// TIA Portal V21 export
ORGANIZATION_BLOCK "Cyclic interrupt"   // OB30, LAD, CyclicInterrupt
{ S7_Optimized_Access := 'TRUE' }
// stored: CyclicTime 5000, SetENOAutomatically false
   VAR_INPUT
      Initial_Call : Bool;
      Event_Count : Int;
   END_VAR
   VAR_TEMP
      virposINT : DInt;
      appo : Real;
      VirOnTarget : Bool;
   END_VAR
   VAR_TEMP   // added for the SCL form of the ladder/FBD networks
      _w1 : Bool;
      _w2 : Bool;
      _w3 : Bool;
      _w4 : Bool;
      _w5 : Bool;
      _w6 : Bool;
   END_VAR
BEGIN

REGION Network 2
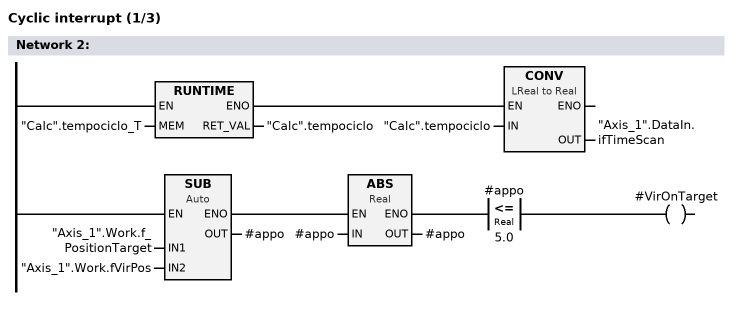
   // no SCL statement known for Runtime: written as a call
   // ENO of a box is taken as its EN; it also drops when the box reports an error
   "Calc".tempociclo := Runtime(mem := "Calc".tempociclo_T);
   "Axis_1".DataIn.ifTimeScan := LREAL_TO_REAL("Calc".tempociclo);
   #appo := "Axis_1".Work.f_PositionTarget - "Axis_1".Work.fVirPos;
   #appo := ABS(#appo);
   #VirOnTarget := #appo <= 5.0;
END_REGION

REGION Network 3
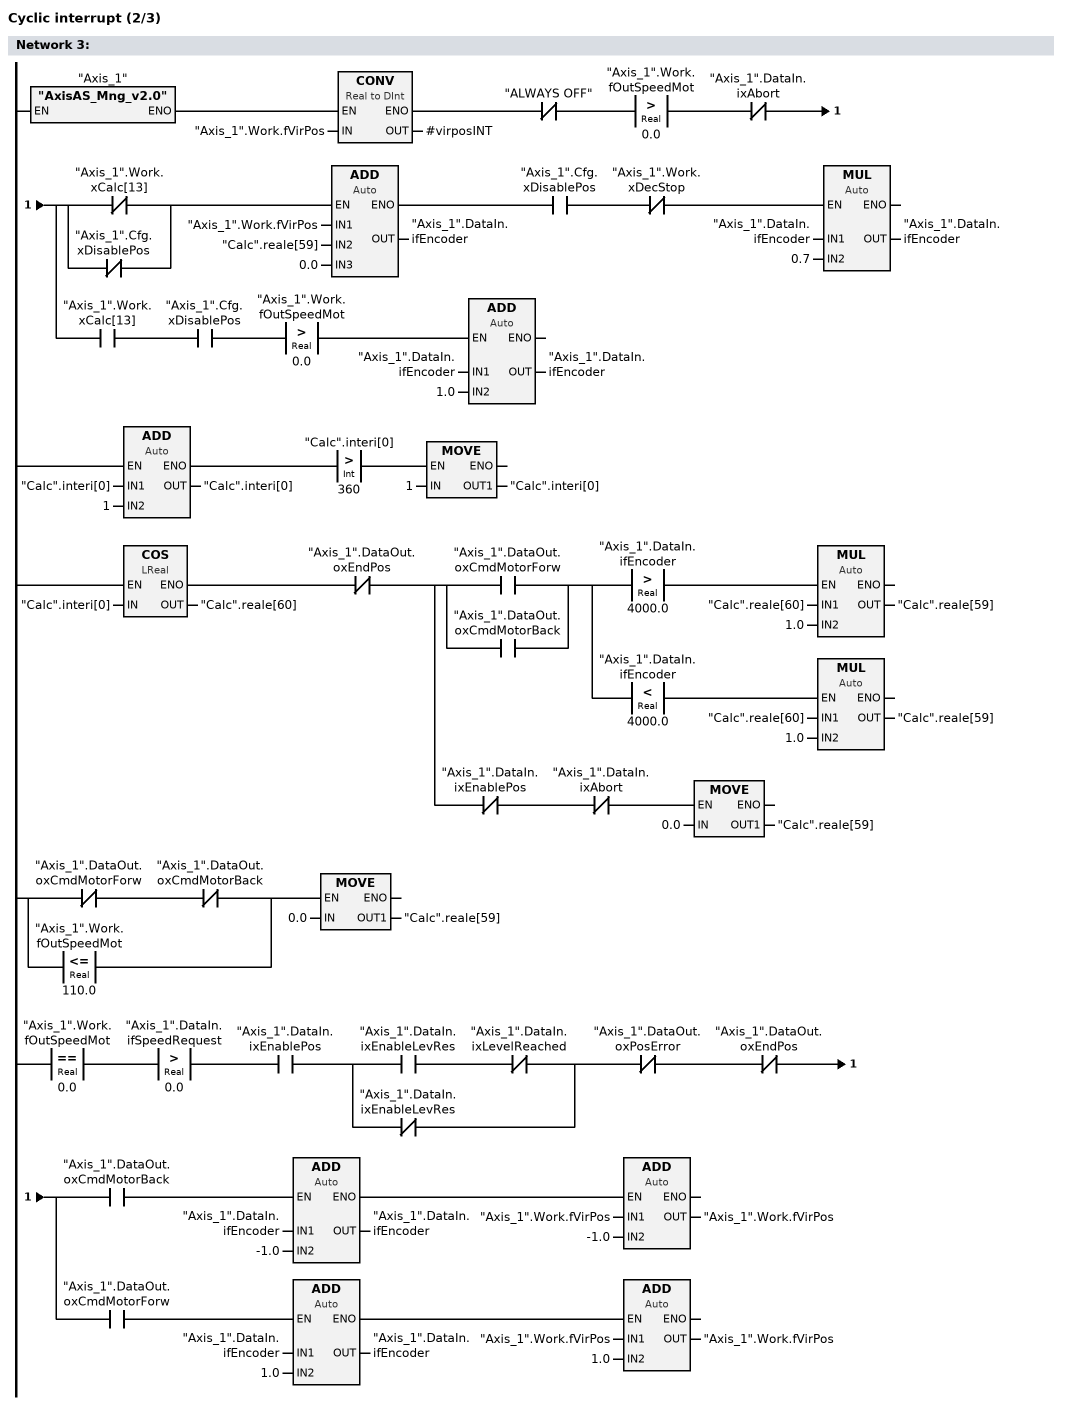
   "Axis_1"(ENO => #_w1);   // "AxisAS_Mng_v2.0"
   IF #_w1 THEN #virposINT := REAL_TO_DINT("Axis_1".Work.fVirPos); END_IF;
   #_w2 := #_w1 AND NOT "ALWAYS OFF" AND ("Axis_1".Work.fOutSpeedMot > 0.0) AND NOT "Axis_1".DataIn.ixAbort;
   #_w3 := #_w2 AND (NOT "Axis_1".Work.xCalc[13] OR NOT "Axis_1".Cfg.xDisablePos);
   IF #_w3 THEN "Axis_1".DataIn.ifEncoder := "Axis_1".Work.fVirPos + "Calc".reale[59] + 0.0; END_IF;
   IF #_w3 AND "Axis_1".Cfg.xDisablePos AND NOT "Axis_1".Work.xDecStop THEN
       "Axis_1".DataIn.ifEncoder := "Axis_1".DataIn.ifEncoder * 0.7;
   END_IF;
   IF #_w2 AND "Axis_1".Work.xCalc[13] AND "Axis_1".Cfg.xDisablePos AND ("Axis_1".Work.fOutSpeedMot > 0.0) THEN
       "Axis_1".DataIn.ifEncoder := "Axis_1".DataIn.ifEncoder + 1.0;
   END_IF;
   "Calc".interi[0] := "Calc".interi[0] + 1;
   IF "Calc".interi[0] > 360 THEN "Calc".interi[0] := 1; END_IF;
   "Calc".reale[60] := COS("Calc".interi[0]);
   #_w4 := NOT "Axis_1".DataOut.oxEndPos;
   #_w5 := #_w4 AND ("Axis_1".DataOut.oxCmdMotorForw OR "Axis_1".DataOut.oxCmdMotorBack);
   IF #_w5 AND ("Axis_1".DataIn.ifEncoder > 4000.0) THEN "Calc".reale[59] := "Calc".reale[60] * 1.0; END_IF;
   IF #_w5 AND ("Axis_1".DataIn.ifEncoder < 4000.0) THEN "Calc".reale[59] := "Calc".reale[60] * 1.0; END_IF;
   IF #_w4 AND NOT "Axis_1".DataIn.ixEnablePos AND NOT "Axis_1".DataIn.ixAbort THEN
       "Calc".reale[59] := 0.0;
   END_IF;
   IF (NOT "Axis_1".DataOut.oxCmdMotorForw AND NOT "Axis_1".DataOut.oxCmdMotorBack) OR ("Axis_1".Work.fOutSpeedMot <= 110.0) THEN
       "Calc".reale[59] := 0.0;
   END_IF;
   #_w6 := ("Axis_1".Work.fOutSpeedMot = 0.0) AND ("Axis_1".DataIn.ifSpeedRequest > 0.0) AND "Axis_1".DataIn.ixEnablePos AND (("Axis_1".DataIn.ixEnableLevRes AND NOT "Axis_1".DataIn.ixLevelReached) OR NOT "Axis_1".DataIn.ixEnableLevRes) AND NOT "Axis_1".DataOut.oxPosError AND NOT "Axis_1".DataOut.oxEndPos;
   IF #_w6 AND "Axis_1".DataOut.oxCmdMotorBack THEN
       "Axis_1".DataIn.ifEncoder := "Axis_1".DataIn.ifEncoder + (-1.0);
       "Axis_1".Work.fVirPos := "Axis_1".Work.fVirPos + (-1.0);
   END_IF;
   IF #_w6 AND "Axis_1".DataOut.oxCmdMotorForw THEN
       "Axis_1".DataIn.ifEncoder := "Axis_1".DataIn.ifEncoder + 1.0;
       "Axis_1".Work.fVirPos := "Axis_1".Work.fVirPos + 1.0;
   END_IF;
END_REGION

REGION Network 4
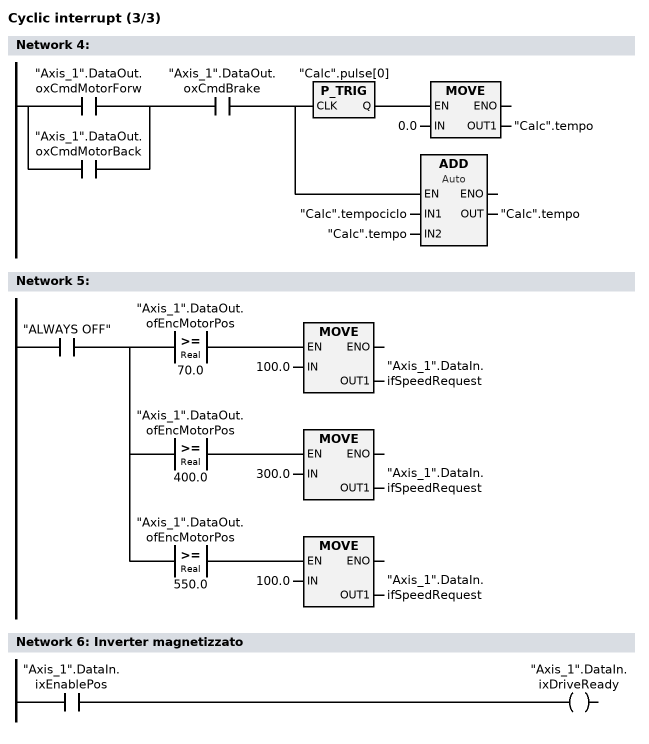
   RUNG wire#powerrail
      Contact( "Axis_1".DataOut.oxCmdMotorForw )
      wire#w1
      Contact( "Axis_1".DataOut.oxCmdBrake )
      wire#w2
      P_Trig( "Calc".pulse[0] )
      Move(in := 0.0, out1 => "Calc".tempo)
   END_RUNG
   RUNG wire#powerrail
      Contact( "Axis_1".DataOut.oxCmdMotorBack )
   END_RUNG wire#w1
   RUNG wire#w2
      Add(in1 := "Calc".tempociclo, in2 := "Calc".tempo, out => "Calc".tempo)
   END_RUNG
   // the same network as SCL:
   #_w1 := ("Axis_1".DataOut.oxCmdMotorForw OR "Axis_1".DataOut.oxCmdMotorBack) AND "Axis_1".DataOut.oxCmdBrake;
   #_w2 := #_w1 AND NOT "Calc".pulse[0];   // rising edge
   "Calc".pulse[0] := #_w1;
   IF #_w2 THEN "Calc".tempo := 0.0; END_IF;
   IF #_w1 THEN "Calc".tempo := "Calc".tempociclo + "Calc".tempo; END_IF;
END_REGION

REGION Network 5
   RUNG wire#powerrail
      Contact( "ALWAYS OFF" )
      wire#w1
      { S7_Templates := "SrcType := Real" } GE_Contact(in1 := "Axis_1".DataOut.ofEncMotorPos, in2 := 70.0)
      Move(in := 100.0, out1 => "Axis_1".DataIn.ifSpeedRequest)
   END_RUNG
   RUNG wire#w1
      { S7_Templates := "SrcType := Real" } GE_Contact(in1 := "Axis_1".DataOut.ofEncMotorPos, in2 := 400.0)
      Move(in := 300.0, out1 => "Axis_1".DataIn.ifSpeedRequest)
   END_RUNG
   RUNG wire#w1
      { S7_Templates := "SrcType := Real" } GE_Contact(in1 := "Axis_1".DataOut.ofEncMotorPos, in2 := 550.0)
      Move(in := 100.0, out1 => "Axis_1".DataIn.ifSpeedRequest)
   END_RUNG
   // the same network as SCL:
   IF "ALWAYS OFF" AND ("Axis_1".DataOut.ofEncMotorPos >= 70.0) THEN
       "Axis_1".DataIn.ifSpeedRequest := 100.0;
   END_IF;
   IF "ALWAYS OFF" AND ("Axis_1".DataOut.ofEncMotorPos >= 400.0) THEN
       "Axis_1".DataIn.ifSpeedRequest := 300.0;
   END_IF;
   IF "ALWAYS OFF" AND ("Axis_1".DataOut.ofEncMotorPos >= 550.0) THEN
       "Axis_1".DataIn.ifSpeedRequest := 100.0;
   END_IF;
END_REGION

REGION Network 6: Inverter magnetizzato
   RUNG wire#powerrail
      Contact( "Axis_1".DataIn.ixEnablePos )
      Coil( "Axis_1".DataIn.ixDriveReady )
   END_RUNG
   // the same network as SCL:
   "Axis_1".DataIn.ixDriveReady := "Axis_1".DataIn.ixEnablePos;
END_REGION
END_ORGANIZATION_BLOCK
